// Mitsubishi GX Developer project: lab 4   PLC: FX1S

PROGRAM MAIN
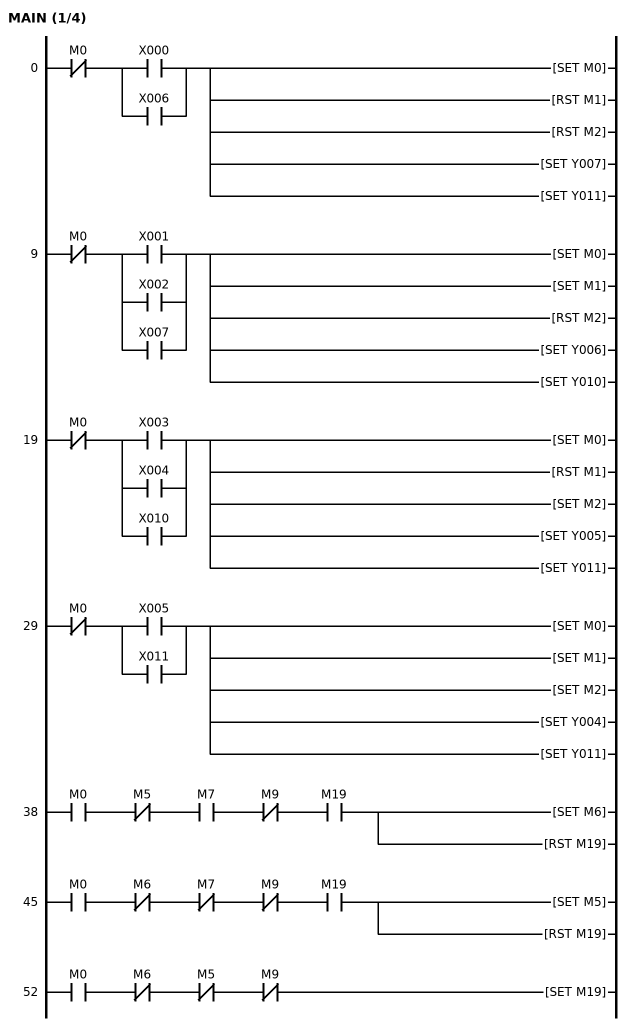
0     LDI     M0
      LD      X000
      OR      X006
      ANB
      SET     M0
      RST     M1
      RST     M2
      SET     Y007
      SET     Y011
9     LDI     M0
      LD      X001
      OR      X002
      OR      X007
      ANB
      SET     M0
      SET     M1
      RST     M2
      SET     Y006
      SET     Y010
19    LDI     M0
      LD      X003
      OR      X004
      OR      X010
      ANB
      SET     M0
      RST     M1
      SET     M2
      SET     Y005
      SET     Y011
29    LDI     M0
      LD      X005
      OR      X011
      ANB
      SET     M0
      SET     M1
      SET     M2
      SET     Y004
      SET     Y011
38    LD      M0
      ANI     M5
      AND     M7
      ANI     M9
      AND     M19
      SET     M6
      RST     M19
45    LD      M0
      ANI     M6
      ANI     M7
      ANI     M9
      AND     M19
      SET     M5
      RST     M19
52    LD      M0
      ANI     M6
      ANI     M5
      ANI     M9
      SET     M19
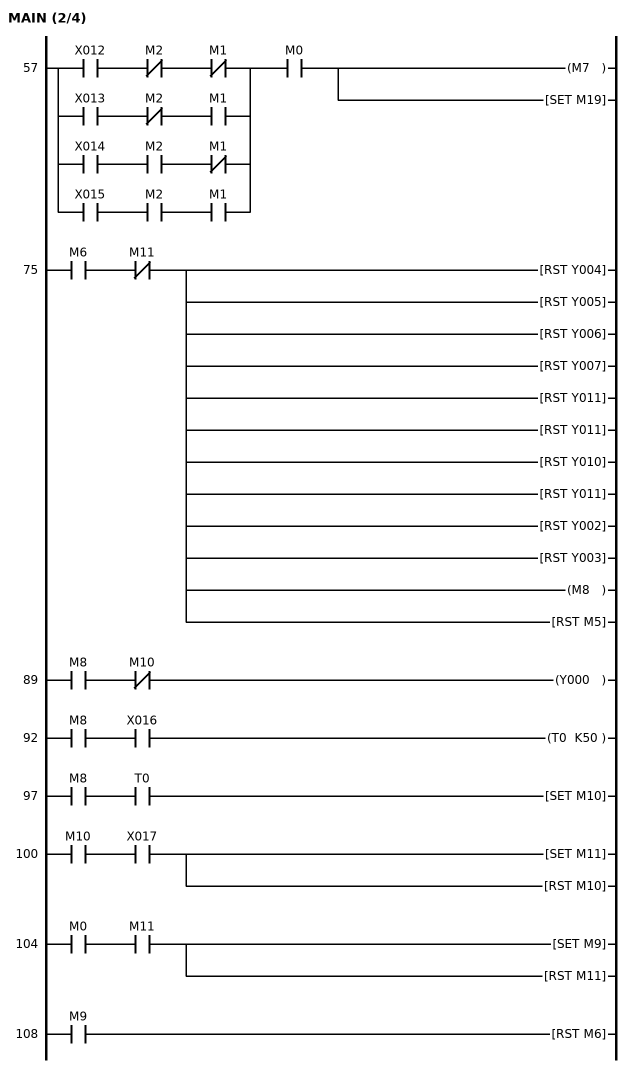
57    LD      X012
      ANI     M2
      ANI     M1
      LD      X013
      ANI     M2
      AND     M1
      ORB
      LD      X014
      AND     M2
      ANI     M1
      ORB
      LD      X015
      AND     M2
      AND     M1
      ORB
      AND     M0
      OUT     M7
      SET     M19
75    LD      M6
      ANI     M11
      RST     Y004
      RST     Y005
      RST     Y006
      RST     Y007
      RST     Y011
      RST     Y011
      RST     Y010
      RST     Y011
      RST     Y002
      RST     Y003
      OUT     M8
      RST     M5
89    LD      M8
      ANI     M10
      OUT     Y000
92    LD      M8
      AND     X016
      OUT     T0 K50
97    LD      M8
      AND     T0
      SET     M10
100   LD      M10
      AND     X017
      SET     M11
      RST     M10
104   LD      M0
      AND     M11
      SET     M9
      RST     M11
108   LD      M9
      RST     M6
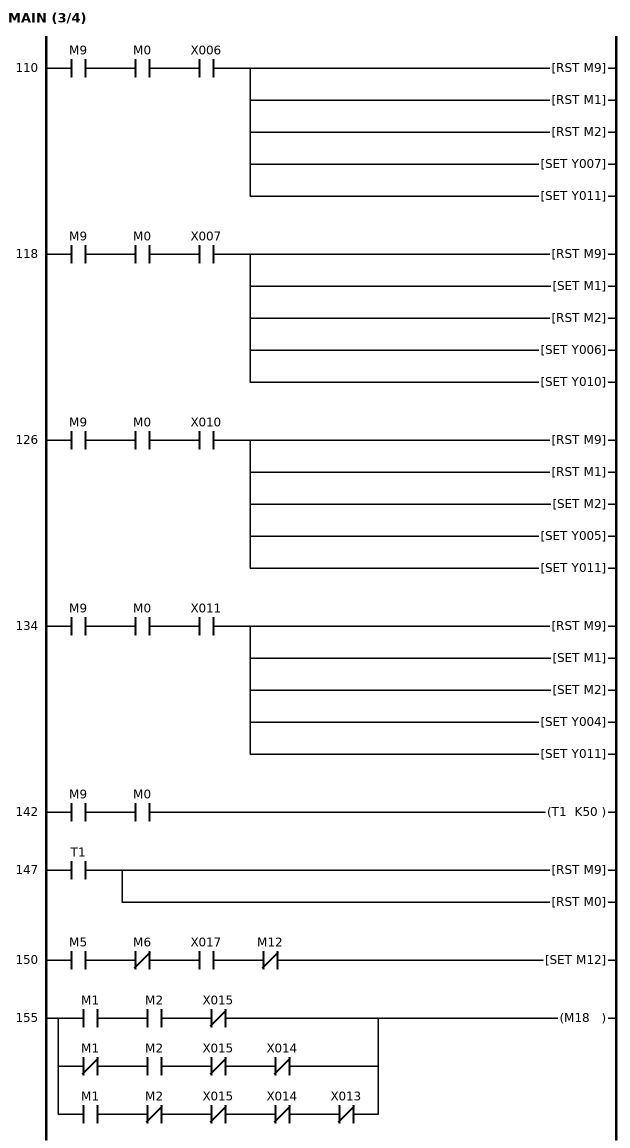
110   LD      M9
      AND     M0
      AND     X006
      RST     M9
      RST     M1
      RST     M2
      SET     Y007
      SET     Y011
118   LD      M9
      AND     M0
      AND     X007
      RST     M9
      SET     M1
      RST     M2
      SET     Y006
      SET     Y010
126   LD      M9
      AND     M0
      AND     X010
      RST     M9
      RST     M1
      SET     M2
      SET     Y005
      SET     Y011
134   LD      M9
      AND     M0
      AND     X011
      RST     M9
      SET     M1
      SET     M2
      SET     Y004
      SET     Y011
142   LD      M9
      AND     M0
      OUT     T1 K50
147   LD      T1
      RST     M9
      RST     M0
150   LD      M5
      ANI     M6
      AND     X017
      ANI     M12
      SET     M12
155   LD      M1
      AND     M2
      ANI     X015
      LDI     M1
      AND     M2
      ANI     X015
      ANI     X014
      ORB
      LD      M1
      ANI     M2
      ANI     X015
      ANI     X014
      ANI     X013
      ORB
      OUT     M18
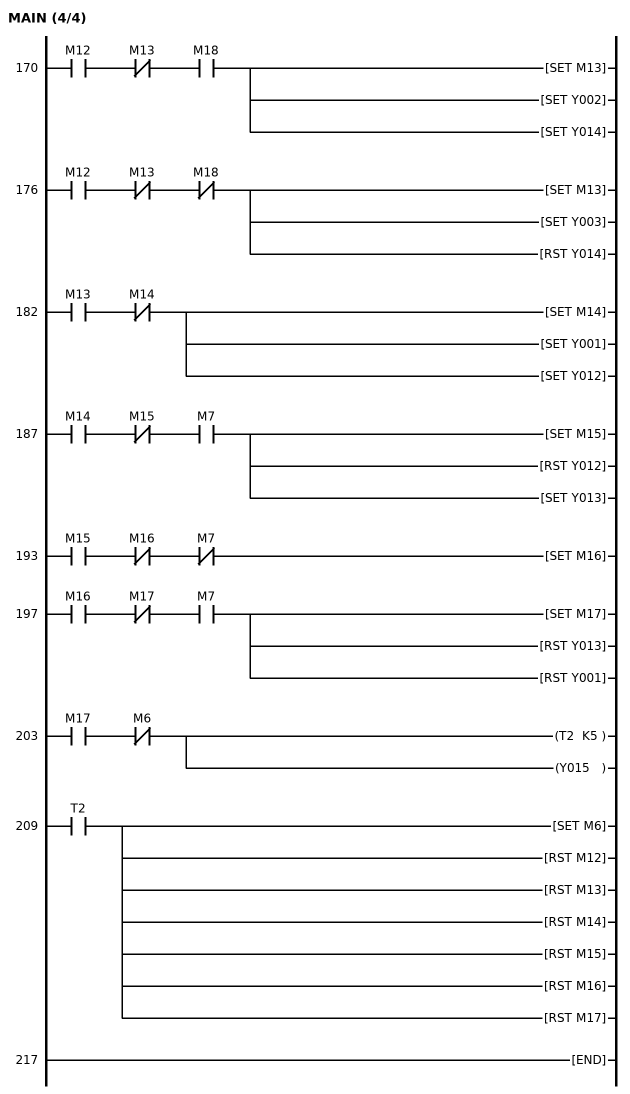
170   LD      M12
      ANI     M13
      AND     M18
      SET     M13
      SET     Y002
      SET     Y014
176   LD      M12
      ANI     M13
      ANI     M18
      SET     M13
      SET     Y003
      RST     Y014
182   LD      M13
      ANI     M14
      SET     M14
      SET     Y001
      SET     Y012
187   LD      M14
      ANI     M15
      AND     M7
      SET     M15
      RST     Y012
      SET     Y013
193   LD      M15
      ANI     M16
      ANI     M7
      SET     M16
197   LD      M16
      ANI     M17
      AND     M7
      SET     M17
      RST     Y013
      RST     Y001
203   LD      M17
      ANI     M6
      OUT     T2 K5
      OUT     Y015
209   LD      T2
      SET     M6
      RST     M12
      RST     M13
      RST     M14
      RST     M15
      RST     M16
      RST     M17
217   END
END_PROGRAM
